Staubli VAL3: string.dtx

mdesc mNomSpeed
public lists lLists
  [0]
    string sString
string sInput[5]
lists lResult
  [0]
    string sString
string sResult
